PROGRAM MAIN
VAR
END_VAR

VAR CONSTANT
	WaterLevMax:		INT:= 200;
	WaterLev3:			INT:= 150;
	WaterLev2:			INT:= 100;
	WaterLev1:			INT:= 50;
END_VAR

(*  function block Washer  *)
(*  2008-10-08  BoS University West *)

(*  -------------  water level  -----------------  *)
IF GVL.ixFill AND GVL.nWaterLev < WaterLevMax THEN				(* increase water level *)
	GVL.nWaterLev := GVL.nWaterLev + 1;
END_IF

IF GVL.ixDrain AND GVL.nWaterLev > 0 THEN						(* decrease water level *)
	GVL.nWaterLev := GVL.nWaterLev - 1;
END_IF

GVL.nShowWater := - GVL.nWaterLev;								(* inverting only for display function *)

(*  -------------  water level sensors  -----------------  *)
IF GVL.nWaterLev > 0 THEN
	GVL.qxNotEmpty := TRUE;
ELSE
	GVL.qxNotEmpty := FALSE;
END_IF
IF GVL.nWaterLev >= WaterLev1 THEN
	GVL.qxLevel1 := TRUE;
ELSE
	GVL.qxLevel1 := FALSE;
END_IF
IF GVL.nWaterLev >= WaterLev2 THEN
	GVL.qxLevel2 := TRUE;
ELSE
	GVL.qxLevel2 := FALSE;
END_IF
IF GVL.nWaterLev >= WaterLev3 THEN
	GVL.qxLevel3 := TRUE;
ELSE
	GVL.qxLevel3 := FALSE;
END_IF

(*  -------------  water temp  -----------------  *)
IF GVL.qxNotEmpty AND GVL.ixHeat AND GVL.nCurTemp < 100 THEN
	GVL.nCurTemp := GVL.nCurTemp + 1;
ELSIF GVL.qxNotEmpty AND NOT GVL.ixHeat AND GVL.nCurTemp > 0 THEN
	GVL.nCurTemp := GVL.nCurTemp - 1;
ELSIF NOT GVL.qxNotEmpty THEN
	GVL.nCurTemp := 20;
END_IF



(*  -------------  water temp sensor  -----------------  *)

IF GVL.nCurTemp > GVL.nSetTemp THEN
	GVL.qxTempOk := TRUE;
ELSE
	GVL.qxTempOk := FALSE;
END_IF

(*  -------------  cylinder posistion  -----------------  *)
IF GVL.ixForw AND NOT GVL.ixSpin THEN
	GVL.nCylPos := GVL.nCylPos+5;
ELSIF GVL.ixForw AND GVL.ixSpin THEN
	GVL.nCylPos := GVL.nCylPos+15;
END_IF
IF GVL.ixBack AND NOT GVL.ixSpin THEN
	GVL.nCylPos := GVL.nCylPos-5;
ELSIF GVL.ixBack AND  GVL.ixSpin THEN
	GVL.nCylPos := GVL.nCylPos-15;
END_IF

IF GVL.nCylPos > 359 THEN
	GVL.nCylPos := 0;
ELSIF GVL.nCylPos < 0 THEN
	GVL.nCylPos :=355;
END_IF

(*  -------------  display number  -----------------  *)
IF NOT GVL.ixDispBit1 AND NOT GVL.ixDispBit2 THEN
	GVL.nDispNo:=0;
ELSIF GVL.ixDispBit1 AND NOT GVL.ixDispBit2 THEN
	GVL.nDispNo:=1;
ELSIF NOT GVL.ixDispBit1 AND  GVL.ixDispBit2 THEN
	GVL.nDispNo:=2;
ELSIF GVL.ixDispBit1 AND GVL.ixDispBit2 THEN
	GVL.nDispNo:=3;
END_IF

END_PROGRAM

(* stored: Version 1.1.0.1, ProductVersion 3.1.4022.12
   POU MAIN: Id {31785a7b-363b-4926-ba76-520e0571d2ce}, SpecialFunc None *)
